(* Logix 5000 project; controller simObli1_rev_1 Emulate 5570 rev 32.11; software revision 32.02; part 2 of 2 *)
(* tags used below, declared in another part *)
   AbsorberingMS1 : SFC_STEP;   // Absorbering MS-1
   Koeling_MS2 : SFC_STEP;   // Køling MS-2 (MS_2 Ladder rung 4 )
   KoelingMS1 : SFC_STEP;   // Køling MS-1,( MS_1 - Ladder ( rung 8)
   OpvarmningMS1 : SFC_STEP;   // Opvarmning MS-1, ( MS_1 Ladder - rung 3)
   OpvarmningMS2 : SFC_STEP;   // Opvarmning MS-2 (MS_2 Ladder rung 1,2,3 )
   TreykreduktionMS2 : SFC_STEP;   // Trykreduktion MS-2 ( MS_2 Ladder - rung 0 )
   TrykreduktionMS1 : SFC_STEP;   // Trykreduktion MS-1 - Ventil V_11 ( MS_1 Ladder - Rung 2)
   TrykstigningMS1 : SFC_STEP;   // Trykstigning MS-1, PT_101 skal stige til 2 bar
   TrykstigningMS2 : SFC_STEP;   // Trykstigning MS-2
   Absorbering_MS2 : SFC_STEP;   // Absorbering_MS2
   AC_1 : BOOL;
   drift : BOOL;
   H1_opvarmer : BOOL;
   Kd : REAL;
   Ki : REAL;
   Kp : REAL;
   Man_auto : BOOL;
   PT_100 : REAL;
   Sp : REAL;
   V_100 : REAL;
   V_101 : BOOL;
   V_102 : BOOL;
   V_103 : BOOL;
   V_104 : BOOL;
   V_105 : REAL;
   V_106 : REAL;
   V_107 : BOOL;
   V_108 : BOOL;
   V_11 : BOOL;
   V_12 : BOOL;
   V_13 : BOOL;
   V_14 : BOOL;
   VMan_101 : BOOL;
   VMan_102 : BOOL;
   VMan_103 : BOOL;
   VMan_104 : BOOL;
   VMan_107 : BOOL;
   VMan_108 : BOOL;
   VMan_11 : BOOL;
   VMan_12 : BOOL;
   VMan_13 : BOOL;
   VMan_14 : BOOL;
(* MS1_2_Function, continued *)

ROUTINE MS1_Ladder   (* ladder *)
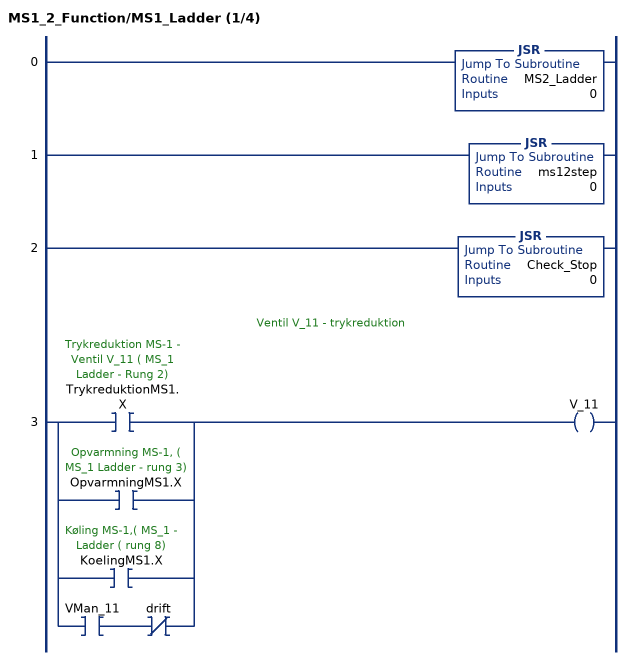
   0: JSR(MS2_Ladder,0);
   1: JSR(ms12step,0);
   2: JSR(Check_Stop,0);
   // Ventil V_11 - trykreduktion
   3: [XIC(TrykreduktionMS1.X) ,XIC(OpvarmningMS1.X) ,XIC(KoelingMS1.X) ,XIC(VMan_11) XIO(drift) ]OTE(V_11);
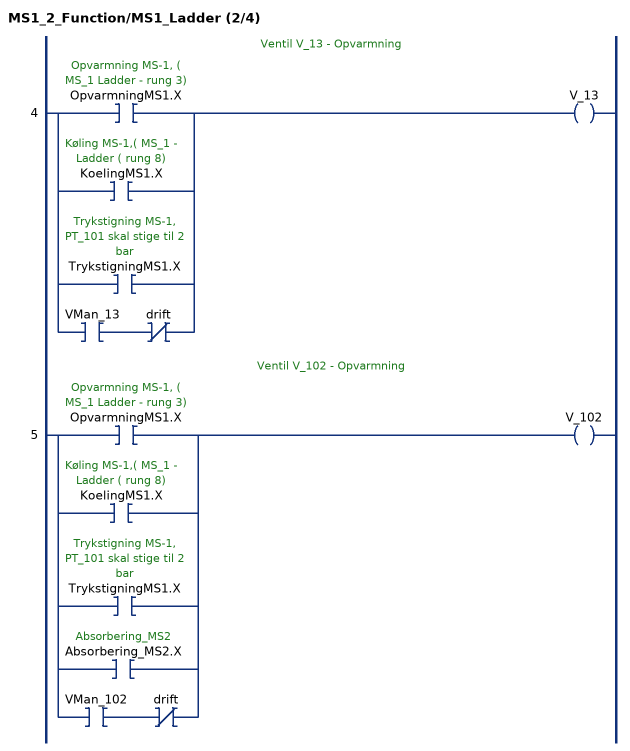
   // Ventil V_13 - Opvarmning
   4: [XIC(OpvarmningMS1.X) ,XIC(KoelingMS1.X) ,XIC(TrykstigningMS1.X) ,XIC(VMan_13) XIO(drift) ]OTE(V_13);
   // Ventil V_102 - Opvarmning
   5: [XIC(OpvarmningMS1.X) ,XIC(KoelingMS1.X) ,XIC(TrykstigningMS1.X) ,XIC(Absorbering_MS2.X) ,XIC(VMan_102) XIO(drift) ]OTE(V_102);
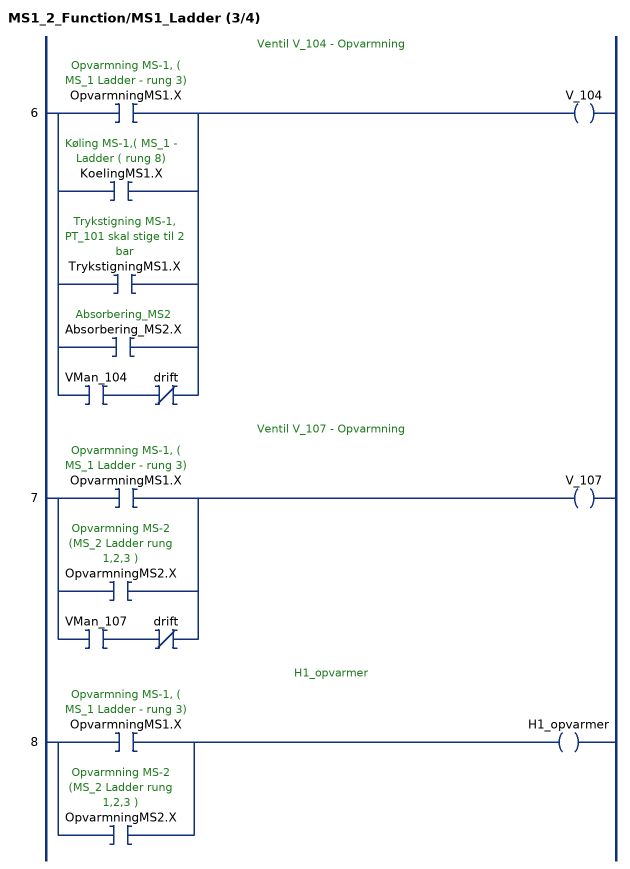
   // Ventil V_104 - Opvarmning
   6: [XIC(OpvarmningMS1.X) ,XIC(KoelingMS1.X) ,XIC(TrykstigningMS1.X) ,XIC(Absorbering_MS2.X) ,XIC(VMan_104) XIO(drift) ]OTE(V_104);
   // Ventil V_107 - Opvarmning
   7: [XIC(OpvarmningMS1.X) ,XIC(OpvarmningMS2.X) ,XIC(VMan_107) XIO(drift) ]OTE(V_107);
   // H1_opvarmer
   8: [XIC(OpvarmningMS1.X) ,XIC(OpvarmningMS2.X) ]OTE(H1_opvarmer);
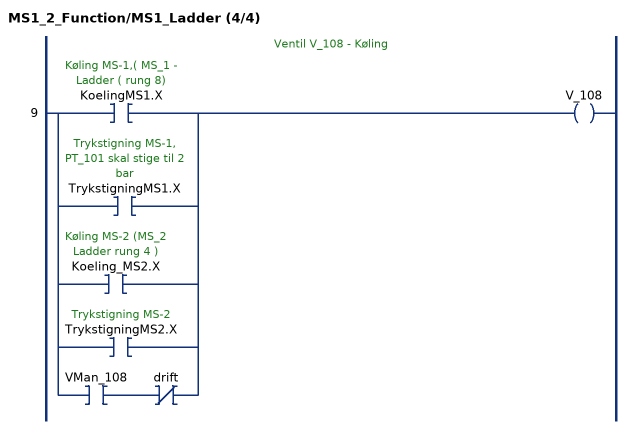
   // Ventil V_108 - Køling
   9: [XIC(KoelingMS1.X) ,XIC(TrykstigningMS1.X) ,XIC(Koeling_MS2.X) ,XIC(TrykstigningMS2.X) ,XIC(VMan_108) XIO(drift) ]OTE(V_108);
END_ROUTINE

ROUTINE MS2_Ladder   (* ladder *)
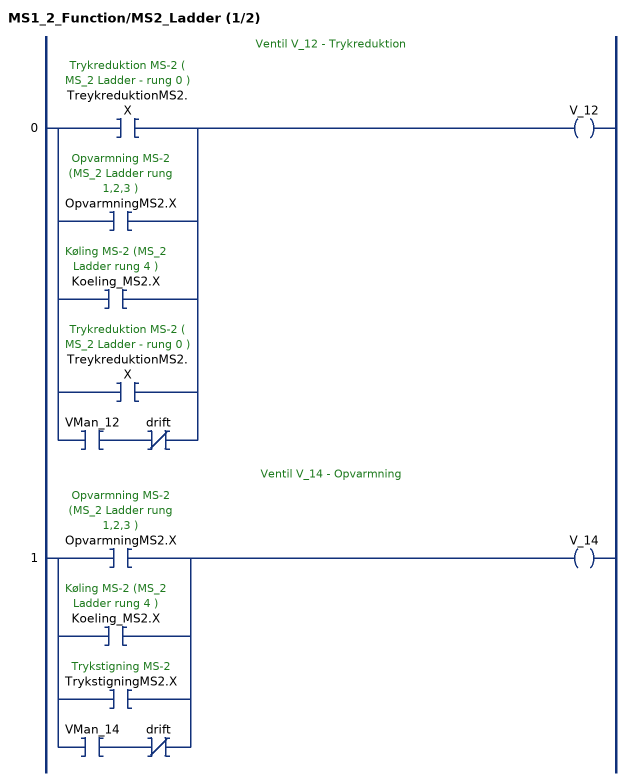
   // Ventil V_12 - Trykreduktion
   0: [XIC(TreykreduktionMS2.X) ,XIC(OpvarmningMS2.X) ,XIC(Koeling_MS2.X) ,XIC(TreykreduktionMS2.X) ,XIC(VMan_12) XIO(drift) ]OTE(V_12);
   // Ventil V_14 - Opvarmning
   1: [XIC(OpvarmningMS2.X) ,XIC(Koeling_MS2.X) ,XIC(TrykstigningMS2.X) ,XIC(VMan_14) XIO(drift) ]OTE(V_14);
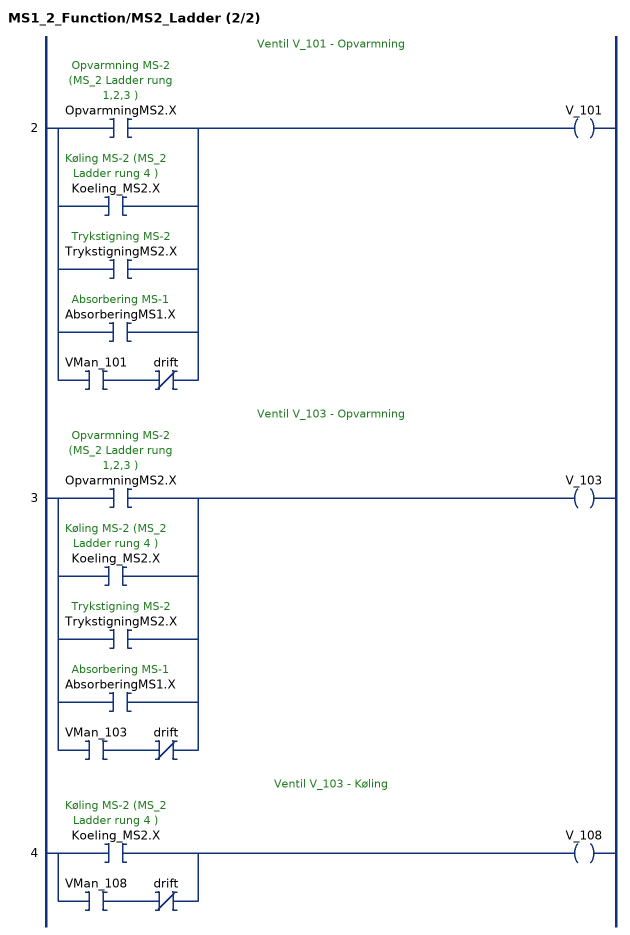
   // Ventil V_101 - Opvarmning
   2: [XIC(OpvarmningMS2.X) ,XIC(Koeling_MS2.X) ,XIC(TrykstigningMS2.X) ,XIC(AbsorberingMS1.X) ,XIC(VMan_101) XIO(drift) ]OTE(V_101);
   // Ventil V_103 - Opvarmning
   3: [XIC(OpvarmningMS2.X) ,XIC(Koeling_MS2.X) ,XIC(TrykstigningMS2.X) ,XIC(AbsorberingMS1.X) ,XIC(VMan_103) XIO(drift) ]OTE(V_103);
   // Ventil V_103 - Køling
   4: [XIC(Koeling_MS2.X) ,XIC(VMan_108) XIO(drift) ]OTE(V_108);
END_ROUTINE

ROUTINE Shutdown   (* structured text *)
// MainTask --> MS1_2_Function
// Slukker for H1-opvarmer, lukker alle ventiler og slukker kompressoren.
   // All valves are closed in First Pass
   // Rutine kan also be run with RESET
   // Globale Tags
   //
   V_11 := 0;
   V_12 := 0;
   V_13 := 0;
   V_14 := 0;
   V_100:= 0; // Also turned off in Trykregulering_PID when drift=0
   V_101 := 0;
   V_102 := 0;
   V_103 := 0;
   V_104 := 0;
   V_105 := 0; // Also turned off in heat_reg when drift = 0
   V_106 := 0; // Also turned of in heat_reg when drift = 0
   V_107 := 0;
   V_108 := 0;
   
   // Turn off heater H1
   H1_opvarmer :=0;
   
   // Turns off compressor AC-1
   AC_1 :=0;
END_ROUTINE
END_PROGRAM

PROGRAM Tryk_regulering_PID   (* main routine PID_Regulator *)
VAR
   BNOT_01 : FBD_BOOLEAN_NOT := (Out := 1);
   PID_regulator_01 : PID_regulator := (SP := 3.0, PV := 1.520366, Kp := 10.0, Ki := 1.0, CV := 14.796341, Manuel_Auto := 1, Reset := 1);
   SCL_01 : SCALE := (InRawMax := 10.0, InEUMax := 100.0, Limiting := 1);
   SEL_01 : SELECT := (In2 := 14.796341);
END_VAR

ROUTINE PID_Regulator   (* function block diagram *)
   SHEET 1
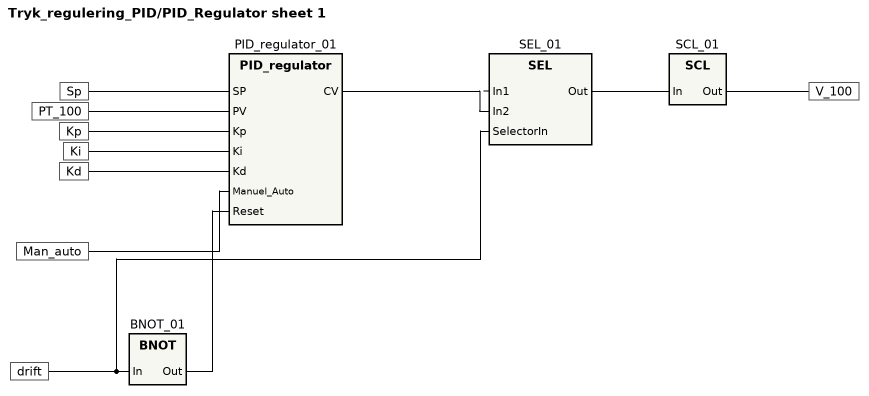
   BNOT_01 : BNOT(In := drift);
   PID_regulator_01 : PID_regulator(SP := Sp, PV := PT_100, Kp := Kp, Ki := Ki, Kd := Kd, Manuel_Auto := Man_auto, Reset := BNOT_01.Out);
   SEL_01 : SEL(In2 := PID_regulator_01.CV, SelectorIn := drift);   // unwired pins: In1
   SCL_01 : SCL(In := SEL_01.Out);
   V_100 := SCL_01.Out;
END_ROUTINE
END_PROGRAM
